{attribute 'qualified_only'}
{attribute 'strict'}
TYPE E_HOME_STATE :
(
	IDLE      := 0,
	RAMP_UP   := 1,
	HOMING    := 2,
	RAMP_DOWN := 3
);
END_TYPE

(* stored: Version 1.1.0.1, ProductVersion 3.1.4024.0
   DUT E_HOME_STATE: Id {321632f8-45eb-4ecd-9713-3f695aaee63b} *)
